// TIA Portal V18 export
FUNCTION_BLOCK "LIVE_BLINK_MONITOR"   // FB65, FBD
{ S7_Optimized_Access := 'TRUE' }
VERSION : 0.1
// stored: AutoNumber true, IsIECCheckEnabled false, IsRetainMemResEnabled false, MemoryReserve 100, SetENOAutomatically false, UDAEnableTagReadback false
   VAR_INPUT
      high_in : Bool;
      flash_in : Bool;
      t_out : Time := T#1s;
      t_resetER : Time := T#5s;
   END_VAR
   VAR_OUTPUT
      ER_no_life : Bool := true;
      remTime : Time;
   END_VAR
   VAR
      tonS { S7_SetPoint := 'True'} : TON_TIME;
      was { S7_SetPoint := 'True'} : Bool;
      tonR { S7_SetPoint := 'True'} : TOF_TIME;
      flashing_ok : Bool;
      flashing_er : Bool;
      high_er : Bool;
   END_VAR
BEGIN

REGION Network 1
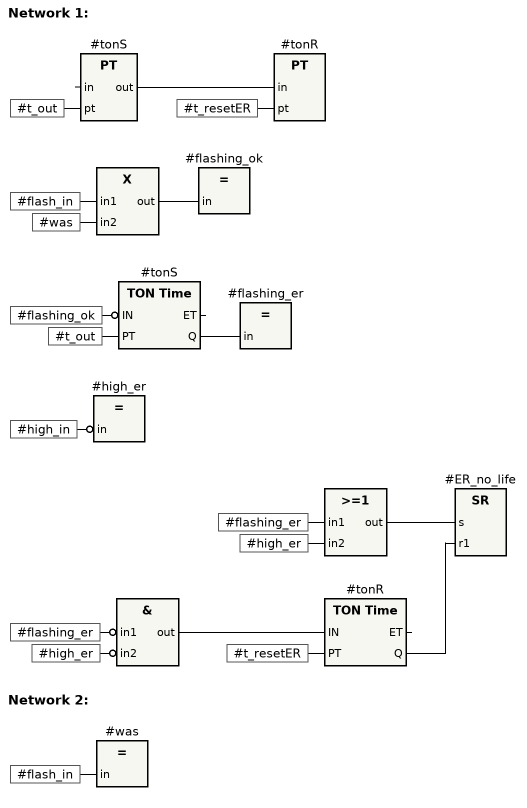
   PRESET_TIMER(PT := #t_out, TIMER := #tonS);
   PRESET_TIMER(PT := #t_resetER, TIMER := #tonR);
   #flashing_ok := #flash_in XOR #was;
   #tonS(IN := NOT #flashing_ok, PT := #t_out);   // TON
   #flashing_er := #tonS.Q;
   #high_er := NOT #high_in;
   #tonR(IN := NOT #flashing_er AND NOT #high_er, PT := #t_resetER);   // TON
   IF #flashing_er OR #high_er THEN
       #ER_no_life := TRUE;   // SR flip-flop
   END_IF;
   IF #tonR.Q THEN #ER_no_life := FALSE; END_IF;
END_REGION

REGION Network 2
   #was := #flash_in;
END_REGION

REGION Network 4 (SCL)
   #remTime := #tonR.PT - #tonR.ET;
END_REGION
END_FUNCTION_BLOCK
